// TIA Portal V15.1 export
// export: Created 2024-06-21T08:41:24.1321259Z, ExportSetting WithDefaults, DisplayName Totally Integrated Automation Portal, DisplayVersion V15.1 Update 5, DisplayName TIA Portal Openness, DisplayVersion V15.1 Update 5, DisplayName SINAMICS Startdrive Advanced, DisplayVersion V15.1, DisplayName G130, G150, S120, S150, SINAMICS MV, S210, DisplayVersion V15.1, DisplayName G110M, G120, G120C, G120D, G120P, DisplayVersion V15.1, DisplayName STEP 7 Professional, DisplayVersion V15.1 Update 5, DisplayName STEP 7 Safety, DisplayVersion V15.1, DisplayName WinCC Professional, DisplayVersion V15.1 Update 5, DisplayName SIMATIC Visualization Architect, DisplayVersion V15.1
FUNCTION "209210ZM01Orders" : Void   // FC303, FBD
TITLE = 209210ZM01Orders
{ S7_Optimized_Access := 'FALSE' }
AUTHOR : VCG
NAME : Mot001
VERSION : 0.1
// stored: AutoNumber false, IsIECCheckEnabled false, SetENOAutomatically False, UDAEnableTagReadback false
   VAR_OUTPUT
      O_AlarmA : Bool;   // Alarm A
      O_AlarmB : Bool;   // Alarm B
      O_AlarmC : Bool;   // Alarm C
      O_AlarmD : Bool;   // Alarm D
      O_AlarmABCondition : Bool;   // Alarms resetable
      H_IAnim : Word;   // Animation bits to Icon in WinCC
   END_VAR
BEGIN

REGION Network 1: **** 4.6 - Machine Status - Indication **** Icon Animation
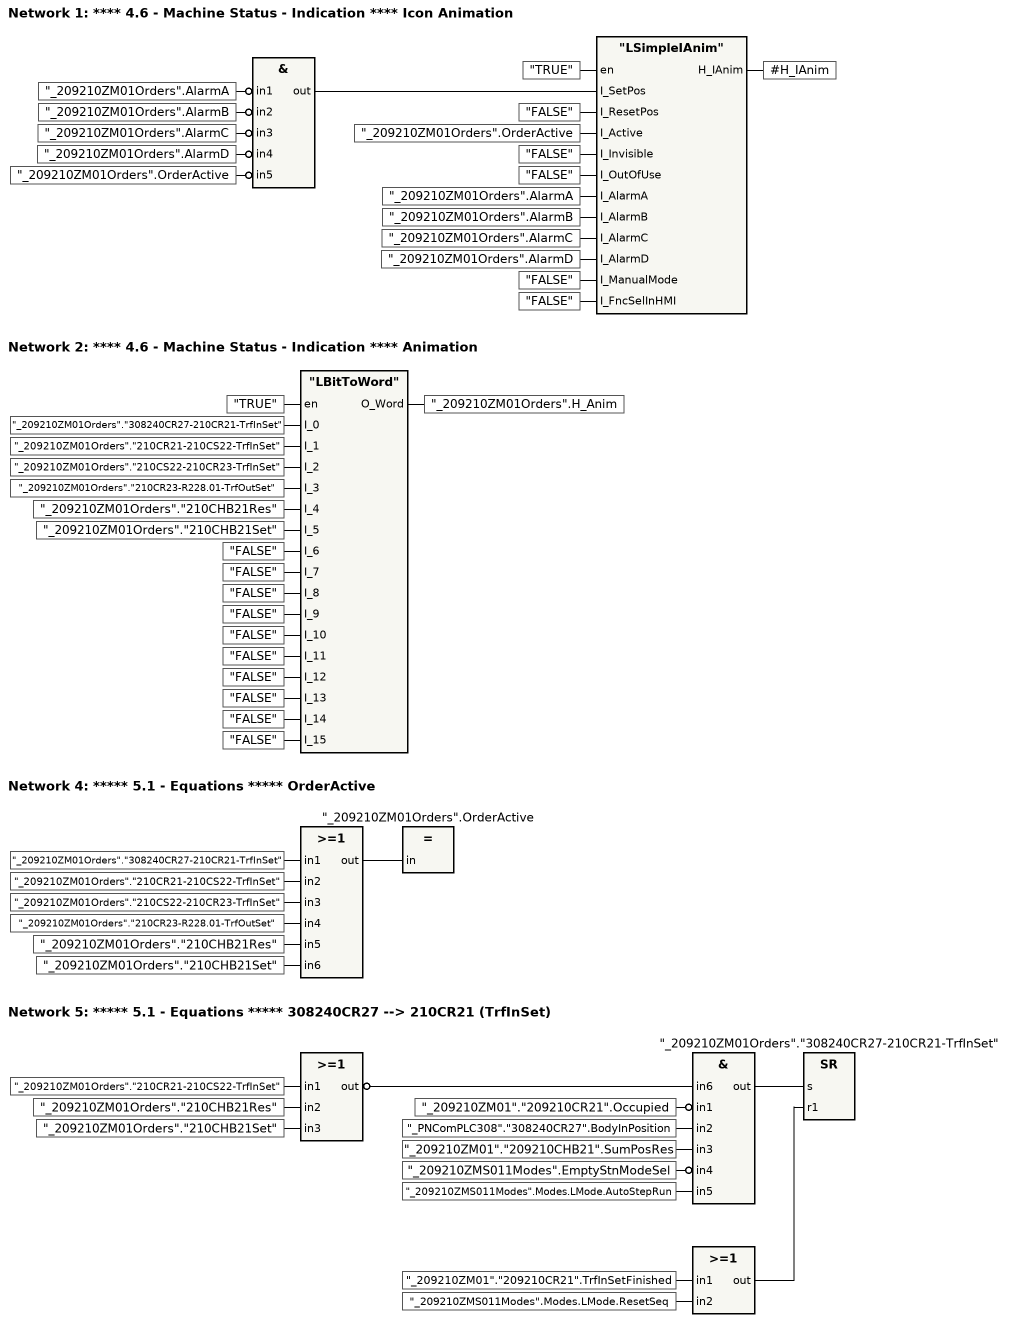
   IF "TRUE" THEN
       "LSimpleIAnim"(I_SetPos := NOT "_209210ZM01Orders".AlarmA AND NOT "_209210ZM01Orders".AlarmB AND NOT "_209210ZM01Orders".AlarmC AND NOT "_209210ZM01Orders".AlarmD AND NOT "_209210ZM01Orders".OrderActive,
                      I_ResetPos := "FALSE",
                      I_Active := "_209210ZM01Orders".OrderActive,
                      I_Invisible := "FALSE",
                      I_OutOfUse := "FALSE",
                      I_AlarmA := "_209210ZM01Orders".AlarmA,
                      I_AlarmB := "_209210ZM01Orders".AlarmB,
                      I_AlarmC := "_209210ZM01Orders".AlarmC,
                      I_AlarmD := "_209210ZM01Orders".AlarmD,
                      I_ManualMode := "FALSE",
                      I_FncSelInHMI := "FALSE",
                      H_IAnim => #H_IAnim);
   END_IF;
END_REGION

REGION Network 2: **** 4.6 - Machine Status - Indication **** Animation
   IF "TRUE" THEN
       "LBitToWord"(I_0 := "_209210ZM01Orders"."308240CR27-210CR21-TrfInSet",
                    I_1 := "_209210ZM01Orders"."210CR21-210CS22-TrfInSet",
                    I_2 := "_209210ZM01Orders"."210CS22-210CR23-TrfInSet",
                    I_3 := "_209210ZM01Orders"."210CR23-R228.01-TrfOutSet",
                    I_4 := "_209210ZM01Orders"."210CHB21Res",
                    I_5 := "_209210ZM01Orders"."210CHB21Set",
                    I_6 := "FALSE",
                    I_7 := "FALSE",
                    I_8 := "FALSE",
                    I_9 := "FALSE",
                    I_10 := "FALSE",
                    I_11 := "FALSE",
                    I_12 := "FALSE",
                    I_13 := "FALSE",
                    I_14 := "FALSE",
                    I_15 := "FALSE",
                    O_Word => "_209210ZM01Orders".H_Anim);
   END_IF;
END_REGION

NETWORK
TITLE = **** 4.6 - Machine Status - Indications **** Animation DB number
// DB number
      OPN   "_209210ZM01Orders";
      L     DBNO;
      T     "_209210ZM01Orders".H_DBnr;

REGION Network 4: ***** 5.1 - Equations ***** OrderActive
   "_209210ZM01Orders".OrderActive := "_209210ZM01Orders"."308240CR27-210CR21-TrfInSet" OR "_209210ZM01Orders"."210CR21-210CS22-TrfInSet" OR "_209210ZM01Orders"."210CS22-210CR23-TrfInSet" OR "_209210ZM01Orders"."210CR23-R228.01-TrfOutSet" OR "_209210ZM01Orders"."210CHB21Res" OR "_209210ZM01Orders"."210CHB21Set";
END_REGION

REGION Network 5: ***** 5.1 - Equations ***** 308240CR27 --> 210CR21 (TrfInSet)
   IF NOT ("_209210ZM01Orders"."210CR21-210CS22-TrfInSet" OR "_209210ZM01Orders"."210CHB21Res" OR "_209210ZM01Orders"."210CHB21Set") AND NOT "_209210ZM01"."209210CR21".Occupied AND "_PNComPLC308"."308240CR27".BodyInPosition AND "_209210ZM01"."209210CHB21".SumPosRes AND NOT "_209210ZMS011Modes".EmptyStnModeSel AND "_209210ZMS011Modes".Modes.LMode.AutoStepRun THEN
       "_209210ZM01Orders"."308240CR27-210CR21-TrfInSet" := TRUE;   // SR flip-flop
   END_IF;
   IF "_209210ZM01"."209210CR21".TrfInSetFinished OR "_209210ZMS011Modes".Modes.LMode.ResetSeq THEN
       "_209210ZM01Orders"."308240CR27-210CR21-TrfInSet" := FALSE;
   END_IF;
END_REGION

REGION Network 6: ***** 5.1 - Equations ***** 210CR21 --> 210CS22 (TrfInSet)
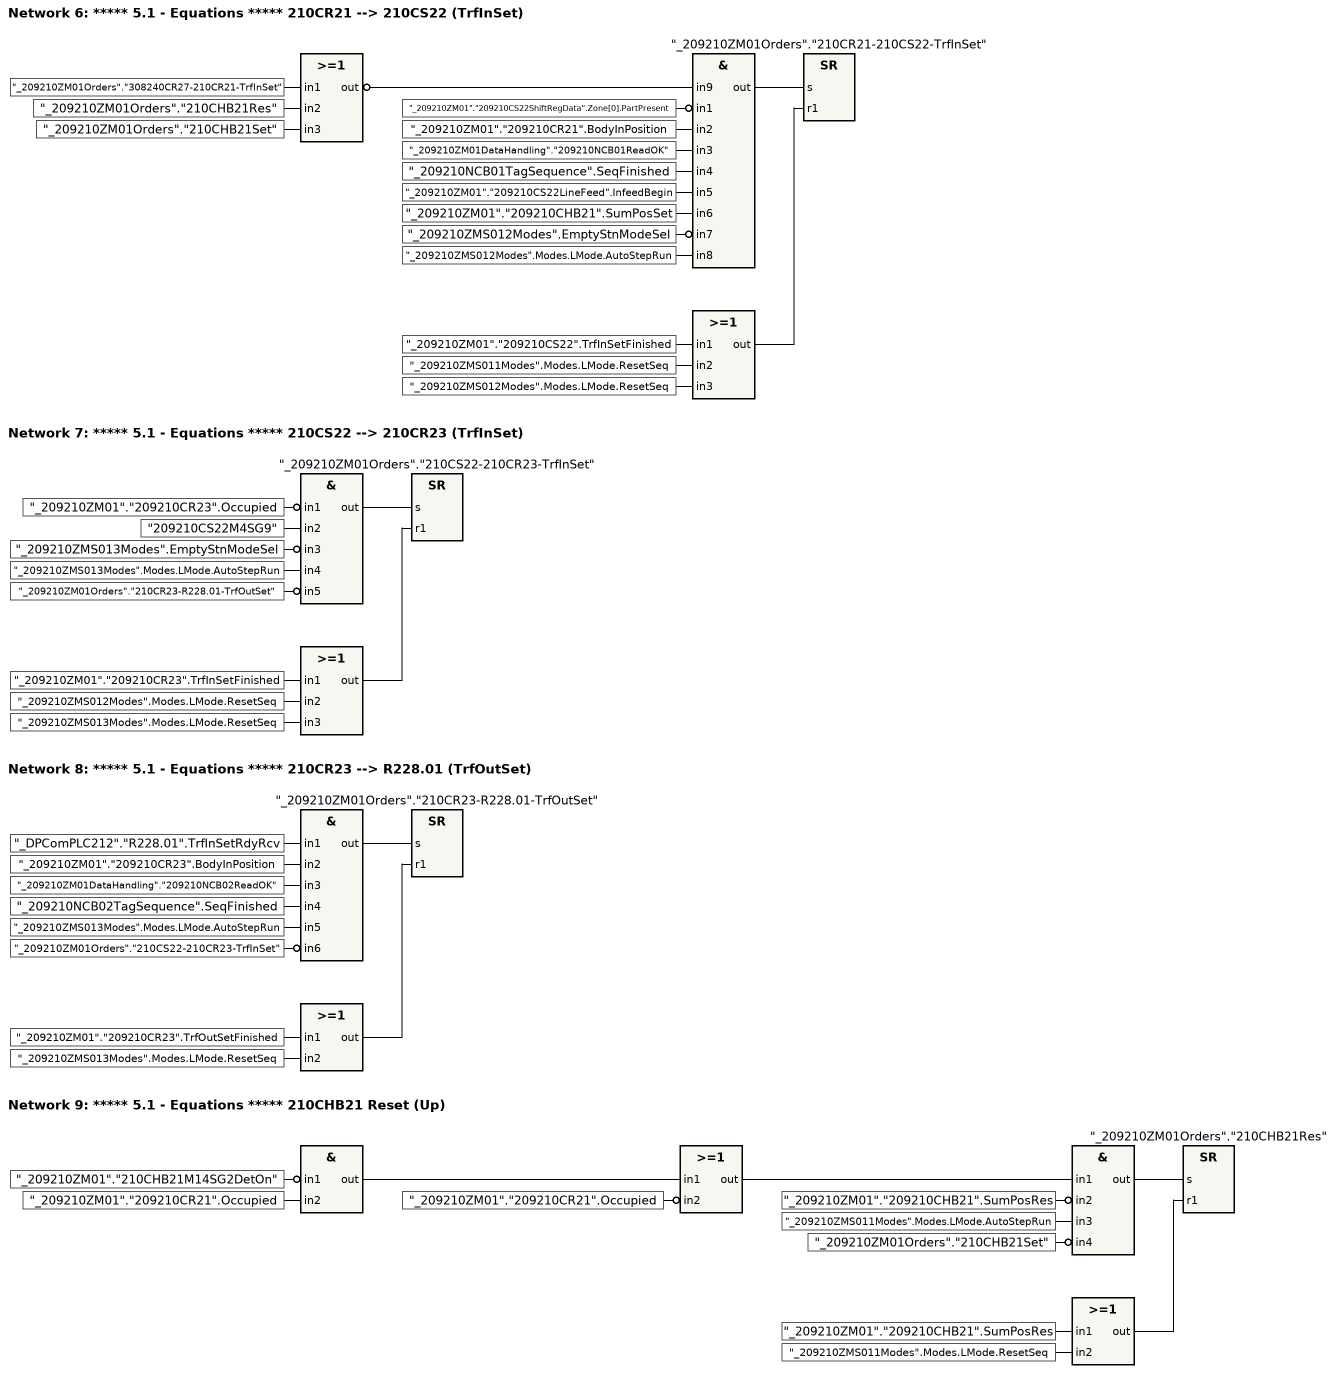
   IF NOT ("_209210ZM01Orders"."308240CR27-210CR21-TrfInSet" OR "_209210ZM01Orders"."210CHB21Res" OR "_209210ZM01Orders"."210CHB21Set") AND NOT "_209210ZM01"."209210CS22ShiftRegData".Zone[0].PartPresent AND "_209210ZM01"."209210CR21".BodyInPosition AND "_209210ZM01DataHandling"."209210NCB01ReadOK" AND "_209210NCB01TagSequence".SeqFinished AND "_209210ZM01"."209210CS22LineFeed".InfeedBegin AND "_209210ZM01"."209210CHB21".SumPosSet AND NOT "_209210ZMS012Modes".EmptyStnModeSel AND "_209210ZMS012Modes".Modes.LMode.AutoStepRun THEN
       "_209210ZM01Orders"."210CR21-210CS22-TrfInSet" := TRUE;   // SR flip-flop
   END_IF;
   IF "_209210ZM01"."209210CS22".TrfInSetFinished OR "_209210ZMS011Modes".Modes.LMode.ResetSeq OR "_209210ZMS012Modes".Modes.LMode.ResetSeq THEN
       "_209210ZM01Orders"."210CR21-210CS22-TrfInSet" := FALSE;
   END_IF;
END_REGION

REGION Network 7: ***** 5.1 - Equations ***** 210CS22 --> 210CR23 (TrfInSet)
   IF NOT "_209210ZM01"."209210CR23".Occupied AND "209210CS22M4SG9" AND NOT "_209210ZMS013Modes".EmptyStnModeSel AND "_209210ZMS013Modes".Modes.LMode.AutoStepRun AND NOT "_209210ZM01Orders"."210CR23-R228.01-TrfOutSet" THEN
       "_209210ZM01Orders"."210CS22-210CR23-TrfInSet" := TRUE;   // SR flip-flop
   END_IF;
   IF "_209210ZM01"."209210CR23".TrfInSetFinished OR "_209210ZMS012Modes".Modes.LMode.ResetSeq OR "_209210ZMS013Modes".Modes.LMode.ResetSeq THEN
       "_209210ZM01Orders"."210CS22-210CR23-TrfInSet" := FALSE;
   END_IF;
END_REGION

REGION Network 8: ***** 5.1 - Equations ***** 210CR23 --> R228.01 (TrfOutSet)
   IF "_DPComPLC212"."R228.01".TrfInSetRdyRcv AND "_209210ZM01"."209210CR23".BodyInPosition AND "_209210ZM01DataHandling"."209210NCB02ReadOK" AND "_209210NCB02TagSequence".SeqFinished AND "_209210ZMS013Modes".Modes.LMode.AutoStepRun AND NOT "_209210ZM01Orders"."210CS22-210CR23-TrfInSet" THEN
       "_209210ZM01Orders"."210CR23-R228.01-TrfOutSet" := TRUE;   // SR flip-flop
   END_IF;
   IF "_209210ZM01"."209210CR23".TrfOutSetFinished OR "_209210ZMS013Modes".Modes.LMode.ResetSeq THEN
       "_209210ZM01Orders"."210CR23-R228.01-TrfOutSet" := FALSE;
   END_IF;
END_REGION

REGION Network 9: ***** 5.1 - Equations ***** 210CHB21 Reset (Up)
   IF ((NOT "_209210ZM01"."210CHB21M14SG2DetOn" AND "_209210ZM01"."209210CR21".Occupied) OR NOT "_209210ZM01"."209210CR21".Occupied) AND NOT "_209210ZM01"."209210CHB21".SumPosRes AND "_209210ZMS011Modes".Modes.LMode.AutoStepRun AND NOT "_209210ZM01Orders"."210CHB21Set" THEN
       "_209210ZM01Orders"."210CHB21Res" := TRUE;   // SR flip-flop
   END_IF;
   IF "_209210ZM01"."209210CHB21".SumPosRes OR "_209210ZMS011Modes".Modes.LMode.ResetSeq THEN
       "_209210ZM01Orders"."210CHB21Res" := FALSE;
   END_IF;
END_REGION

REGION Network 10: ***** 5.1 - Equations ***** 210CHB21 Set (Down)
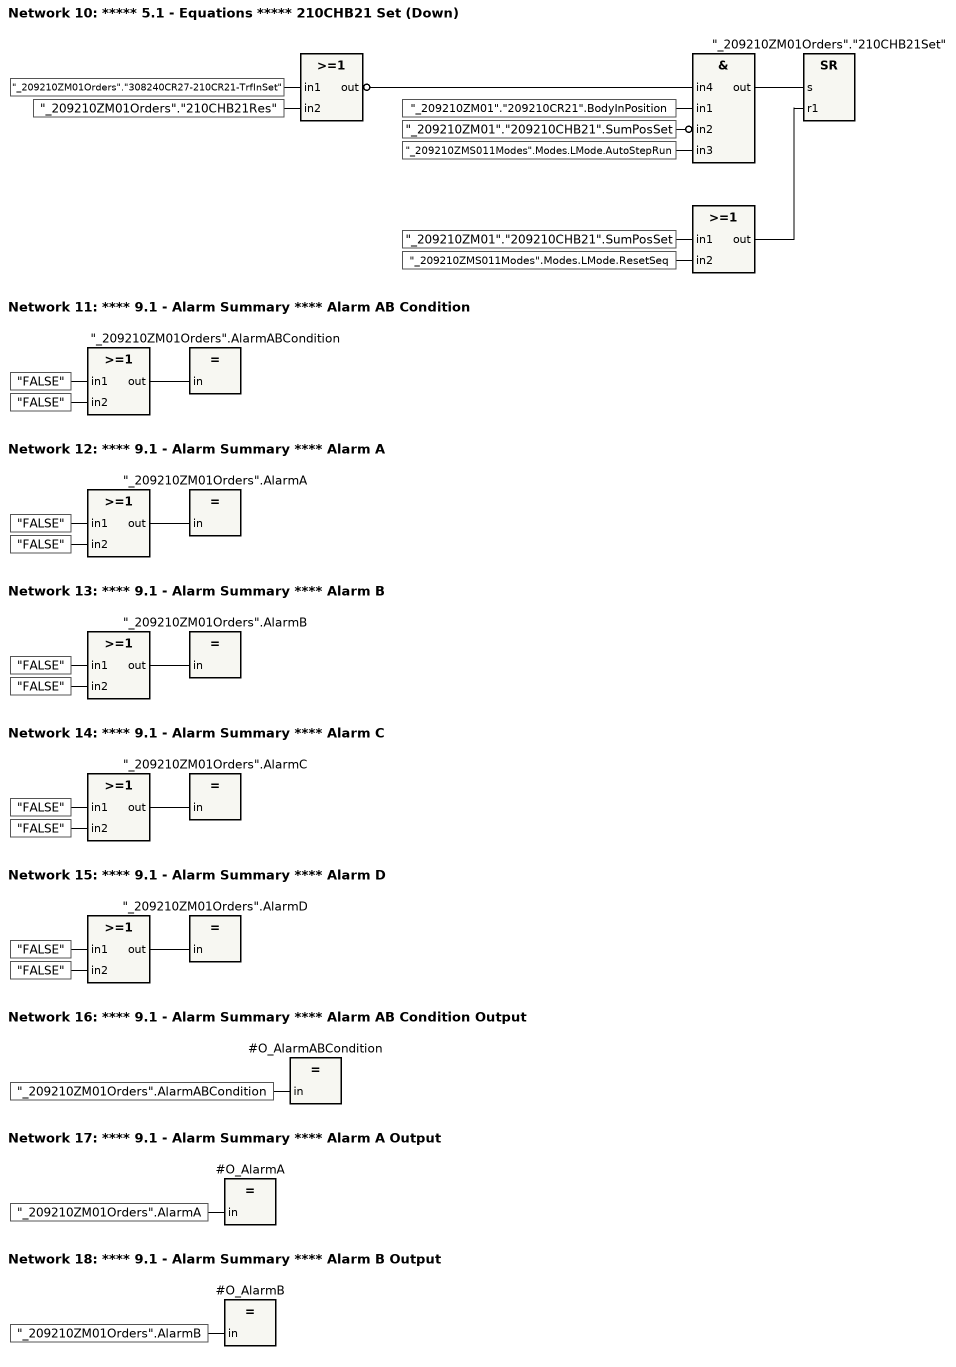
   IF NOT ("_209210ZM01Orders"."308240CR27-210CR21-TrfInSet" OR "_209210ZM01Orders"."210CHB21Res") AND "_209210ZM01"."209210CR21".BodyInPosition AND NOT "_209210ZM01"."209210CHB21".SumPosSet AND "_209210ZMS011Modes".Modes.LMode.AutoStepRun THEN
       "_209210ZM01Orders"."210CHB21Set" := TRUE;   // SR flip-flop
   END_IF;
   IF "_209210ZM01"."209210CHB21".SumPosSet OR "_209210ZMS011Modes".Modes.LMode.ResetSeq THEN
       "_209210ZM01Orders"."210CHB21Set" := FALSE;
   END_IF;
END_REGION

REGION Network 11: **** 9.1 - Alarm Summary **** Alarm AB Condition
   "_209210ZM01Orders".AlarmABCondition := "FALSE" OR "FALSE";
END_REGION

REGION Network 12: **** 9.1 - Alarm Summary **** Alarm A
   "_209210ZM01Orders".AlarmA := "FALSE" OR "FALSE";
END_REGION

REGION Network 13: **** 9.1 - Alarm Summary **** Alarm B
   "_209210ZM01Orders".AlarmB := "FALSE" OR "FALSE";
END_REGION

REGION Network 14: **** 9.1 - Alarm Summary **** Alarm C
   "_209210ZM01Orders".AlarmC := "FALSE" OR "FALSE";
END_REGION

REGION Network 15: **** 9.1 - Alarm Summary **** Alarm D
   "_209210ZM01Orders".AlarmD := "FALSE" OR "FALSE";
END_REGION

REGION Network 16: **** 9.1 - Alarm Summary **** Alarm AB Condition Output
   #O_AlarmABCondition := "_209210ZM01Orders".AlarmABCondition;
END_REGION

REGION Network 17: **** 9.1 - Alarm Summary **** Alarm A Output
   #O_AlarmA := "_209210ZM01Orders".AlarmA;
END_REGION

REGION Network 18: **** 9.1 - Alarm Summary **** Alarm B Output
   #O_AlarmB := "_209210ZM01Orders".AlarmB;
END_REGION

REGION Network 19: **** 9.1 - Alarm Summary **** Alarm C Output
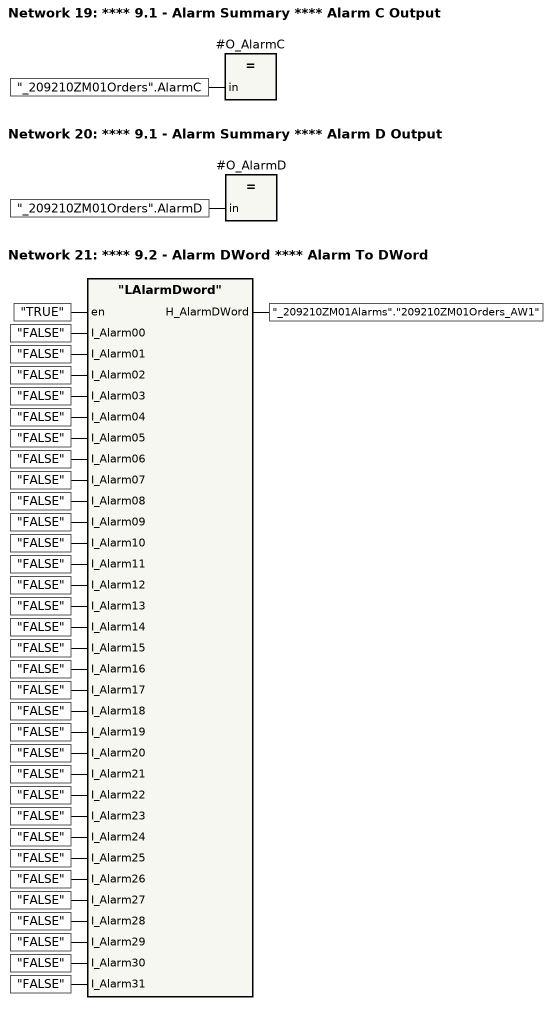
   #O_AlarmC := "_209210ZM01Orders".AlarmC;
END_REGION

REGION Network 20: **** 9.1 - Alarm Summary **** Alarm D Output
   #O_AlarmD := "_209210ZM01Orders".AlarmD;
END_REGION

REGION Network 21: **** 9.2 - Alarm DWord **** Alarm To DWord
   // Alarm Word
   IF "TRUE" THEN
       "LAlarmDword"(I_Alarm00 := "FALSE",
                     I_Alarm01 := "FALSE",
                     I_Alarm02 := "FALSE",
                     I_Alarm03 := "FALSE",
                     I_Alarm04 := "FALSE",
                     I_Alarm05 := "FALSE",
                     I_Alarm06 := "FALSE",
                     I_Alarm07 := "FALSE",
                     I_Alarm08 := "FALSE",
                     I_Alarm09 := "FALSE",
                     I_Alarm10 := "FALSE",
                     I_Alarm11 := "FALSE",
                     I_Alarm12 := "FALSE",
                     I_Alarm13 := "FALSE",
                     I_Alarm14 := "FALSE",
                     I_Alarm15 := "FALSE",
                     I_Alarm16 := "FALSE",
                     I_Alarm17 := "FALSE",
                     I_Alarm18 := "FALSE",
                     I_Alarm19 := "FALSE",
                     I_Alarm20 := "FALSE",
                     I_Alarm21 := "FALSE",
                     I_Alarm22 := "FALSE",
                     I_Alarm23 := "FALSE",
                     I_Alarm24 := "FALSE",
                     I_Alarm25 := "FALSE",
                     I_Alarm26 := "FALSE",
                     I_Alarm27 := "FALSE",
                     I_Alarm28 := "FALSE",
                     I_Alarm29 := "FALSE",
                     I_Alarm30 := "FALSE",
                     I_Alarm31 := "FALSE",
                     H_AlarmDWord => "_209210ZM01Alarms"."209210ZM01Orders_AW1");
   END_IF;
END_REGION
END_FUNCTION
